PROGRAM MAIN
VAR
    {attribute 'OPC.UA.DA':='1'}
    fbTelescope : FB_AsaTelescope( 
          // sTelHost := '10.33.179.130', nTelPort := 11111, sAccHost := 'localhost', nAccPort := 11112); // Leuven
             sTelHost := 'localhost', nTelPort := 32323, sAccHost := 'localhost', nAccPort := 32323); // Simulator
END_VAR

fbTelescope();

END_PROGRAM

(* stored: Version 1.1.0.1, ProductVersion 3.1.4024.12
   POU MAIN: Id {e547a803-3a78-4e51-83ae-77d801307806}, SpecialFunc None *)
